PROGRAM MAIN
VAR

	fbKeuken: TP := (PT := TIME#60ms);
	bKeuken AT %i*: BOOL := false;
	bLED1 AT %Q*: BOOL := false;
END_VAR

fbKeuken(IN:= bKeuken , Q=>bLED1);

END_PROGRAM

(* stored: Version 1.1.0.1, ProductVersion 3.1.4024.12
   POU MAIN: Id {f4168cb9-de31-4179-bb1b-29edc09c54f1}, SpecialFunc None *)
